PROGRAM PB_TestRunner
VAR
    TestSuite_AdsTests : TestSuite_AdsTests;
END_VAR

TestSuite_AdsTests();

END_PROGRAM

(* stored: Version 1.1.0.1, ProductVersion 3.1.4024.12
   POU PB_TestRunner: Id {fa6e722f-1558-004a-1db2-3e3393d796db}, SpecialFunc None *)
